DATA_BLOCK "Zne05_DB"
{ S7_Optimized_Access := 'TRUE' }
VERSION : 0.1
NON_RETAIN
"Zne05"

BEGIN

END_DATA_BLOCK

